// TIA Portal project "FactoryIO_Template_S7-1200_V16_V16" (V16)
// Vorlageprojekt für das Buch mit Zielsystem S7-1200

(* hardware
DEVICE "S7-1200-Station_1"  S7-1200 Station
   slot 0: "Baugruppenträger_0"  Rack  V1.0
   slot 1: "PLC_1"  CPU 1211C DC/DC/DC  6ES7 211-1AE40-0XB0  V4.1
*)

// ===== PLC "PLC_1"  CPU 1211C DC/DC/DC =====

VAR_GLOBAL   // PLC tag table "Standard-Variablentabelle"
   "Tag_1" AT %M0.0 : Bool;
   "Tag_2" AT %M0.1 : Bool;
   "Tag_3" AT %M0.2 : Bool;
   "Tag_4" AT %M0.3 : Bool;
   "Tag_5" AT %M0.4 : Bool;
   "Tag_6" AT %M0.5 : Bool;
   "Tag_7" AT %M1.0 : Bool;
   "Tag_8" AT %M0.6 : Bool;
   "Tag_9" AT %M1.2 : Bool;
   "Tag_10" AT %M1.5 : Bool;
   "Tag_11" AT %M0.7 : Bool;
END_VAR

VAR_GLOBAL   // PLC tag table "Tag table_1"
   "start" AT %I0.0 : Bool;
   "stop" AT %I0.1 : Bool;
   "sen 1" AT %I0.2 : Bool;
   "sen2" AT %I0.3 : Bool;
   "sen 3" AT %I0.4 : Bool;
   "sen4" AT %I0.5 : Bool;
   "sen 5" AT %I0.6 : Bool;
   "detect" AT %I0.7 : Bool;
   "X moving" AT %I1.0 : Bool;
   "Z moving" AT %I1.1 : Bool;
   "curve" AT %Q0.0 : Bool;
   "belt 4" AT %Q0.1 : Bool;
   "belt 6" AT %Q0.2 : Bool;
   "X" AT %Q0.3 : Bool;
   "Z" AT %Q0.4 : Bool;
   "grab" AT %Q0.5 : Bool;
END_VAR

FUNCTION "MHJ-PLC-Lab-Function-S71200" : Void   // FC9000, SCL
{ S7_Optimized_Access := 'TRUE' }
VERSION : 0.1
   VAR_TEMP
      rdTimeReturn : Int;
      outputTime : DTL;
      SyncVal : Byte;
      forVal : Int;
      forVal_2 : Int;
      Value : Byte;
   END_VAR
   VAR CONSTANT
      CompVal : Byte := 16#34;
      Value_01 : Byte := 16#11;
      Value_01_DW : DWord := 16#A165_D992;
      Value_02_DW : DWord := 16#58BE_4401;
   END_VAR
BEGIN

   #Value:=PEEK(area := 16#82,
        dbNumber := 0,
        byteOffset := 511);
   #Value := #Value + 1;

   POKE(area := 16#82,
        dbNumber := 0,
        byteOffset := 511,
        value := #Value);

   POKE(area:=16#81,
        dbNumber:=0,
        byteOffset:=1016,
        value:=#Value_01_DW);
   POKE(area := 16#81,
        dbNumber := 0,
        byteOffset := 1020,
        value := #Value_02_DW);

   POKE(area := 16#81,
        dbNumber := 0,
        byteOffset := 511,
        value := B#16#00);

   FOR #forVal := 0 TO 120 DO
       FOR #forVal_2:=0 TO 10 DO
           #rdTimeReturn:=RD_SYS_T(#outputTime);
           #rdTimeReturn := WR_SYS_T(#outputTime);
           #rdTimeReturn := RD_SYS_T(#outputTime);
           #rdTimeReturn := WR_SYS_T(#outputTime);
       END_FOR;
       #SyncVal:= PEEK(area := 16#81,
                      dbNumber := 0,
                      byteOffset := 511);
       IF #SyncVal = #CompVal THEN
          GOTO M_1;
       END_IF;
   END_FOR;
   RETURN;

   M_1:
   POKE(area := 16#81,
        dbNumber := 0,
        byteOffset := 511,
        value := B#16#0);
END_FUNCTION

ORGANIZATION_BLOCK "Main"   // OB1, LAD, ProgramCycle
TITLE = "Main Program Sweep (Cycle)"
{ S7_Optimized_Access := 'TRUE' }
VERSION : 0.1
   VAR_INPUT
      Initial_Call : Bool;   // Initial call of this OB
      Remanence : Bool;   // =True, if remanent data are available
   END_VAR
   VAR_TEMP   // added for the SCL form of the ladder/FBD networks
      _w1 : Bool;
   END_VAR
BEGIN

REGION Network 1: Konnektierungsbaustein für PLC-Lab
   // Im Netzwerk 1 wird der Konnektierungsbaustein für PLC-Lab aufgerufen.
   // Dieser Aufruf darf nicht entfernt werden!
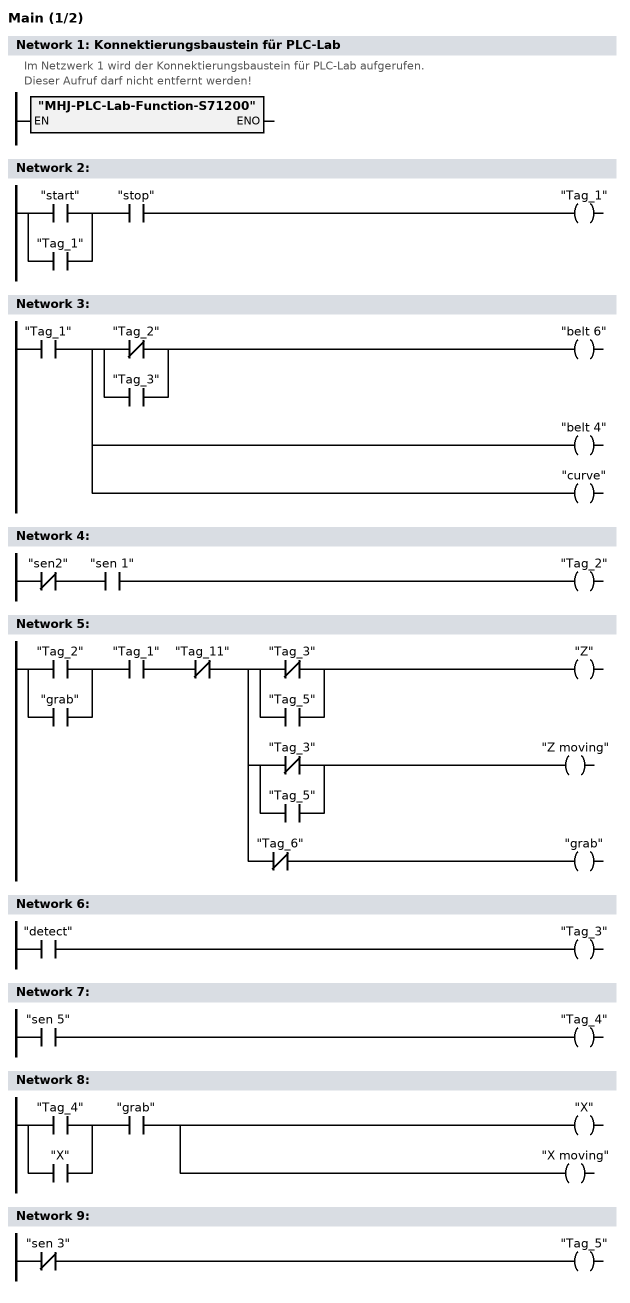
   RUNG wire#powerrail
      "MHJ-PLC-Lab-Function-S71200"()
   END_RUNG
   // the same network as SCL:
   "MHJ-PLC-Lab-Function-S71200"();
END_REGION

REGION Network 2
   RUNG wire#powerrail
      Contact( "start" )
      wire#w1
      Contact( "stop" )
      Coil( "Tag_1" )
   END_RUNG
   RUNG wire#powerrail
      Contact( "Tag_1" )
   END_RUNG wire#w1
   // the same network as SCL:
   "Tag_1" := ("start" OR "Tag_1") AND "stop";
END_REGION

REGION Network 3
   RUNG wire#powerrail
      Contact( "Tag_1" )
      wire#w1
      I_Contact( "Tag_2" )
      wire#w2
      Coil( "belt 6" )
   END_RUNG
   RUNG wire#w1
      Contact( "Tag_3" )
   END_RUNG wire#w2
   RUNG wire#w1
      Coil( "belt 4" )
   END_RUNG
   RUNG wire#w1
      Coil( "curve" )
   END_RUNG
   // the same network as SCL:
   "belt 6" := "Tag_1" AND (NOT "Tag_2" OR "Tag_3");
   "belt 4" := "Tag_1";
   "curve" := "Tag_1";
END_REGION

REGION Network 4
   RUNG wire#powerrail
      I_Contact( "sen2" )
      Contact( "sen 1" )
      Coil( "Tag_2" )
   END_RUNG
   // the same network as SCL:
   "Tag_2" := NOT "sen2" AND "sen 1";
END_REGION

REGION Network 5
   RUNG wire#powerrail
      Contact( "Tag_2" )
      wire#w1
      Contact( "Tag_1" )
      I_Contact( "Tag_11" )
      wire#w2
      I_Contact( "Tag_3" )
      wire#w3
      Coil( "Z" )
   END_RUNG
   RUNG wire#powerrail
      Contact( "grab" )
   END_RUNG wire#w1
   RUNG wire#w2
      Contact( "Tag_5" )
   END_RUNG wire#w3
   RUNG wire#w2
      I_Contact( "Tag_3" )
      wire#w4
      Coil( "Z moving" )
   END_RUNG
   RUNG wire#w2
      Contact( "Tag_5" )
   END_RUNG wire#w4
   RUNG wire#w2
      I_Contact( "Tag_6" )
      Coil( "grab" )
   END_RUNG
   // the same network as SCL:
   #_w1 := ("Tag_2" OR "grab") AND "Tag_1" AND NOT "Tag_11";
   "Z" := #_w1 AND (NOT "Tag_3" OR "Tag_5");
   "Z moving" := #_w1 AND (NOT "Tag_3" OR "Tag_5");
   "grab" := #_w1 AND NOT "Tag_6";
END_REGION

REGION Network 6
   RUNG wire#powerrail
      Contact( "detect" )
      Coil( "Tag_3" )
   END_RUNG
   // the same network as SCL:
   "Tag_3" := "detect";
END_REGION

REGION Network 7
   RUNG wire#powerrail
      Contact( "sen 5" )
      Coil( "Tag_4" )
   END_RUNG
   // the same network as SCL:
   "Tag_4" := "sen 5";
END_REGION

REGION Network 8
   RUNG wire#powerrail
      Contact( "Tag_4" )
      wire#w1
      Contact( "grab" )
      wire#w2
      Coil( "X" )
   END_RUNG
   RUNG wire#powerrail
      Contact( "X" )
   END_RUNG wire#w1
   RUNG wire#w2
      Coil( "X moving" )
   END_RUNG
   // the same network as SCL:
   "X" := ("Tag_4" OR "X") AND "grab";
   "X moving" := "X";
END_REGION

REGION Network 9
   RUNG wire#powerrail
      I_Contact( "sen 3" )
      Coil( "Tag_5" )
   END_RUNG
   // the same network as SCL:
   "Tag_5" := NOT "sen 3";
END_REGION

REGION Network 10
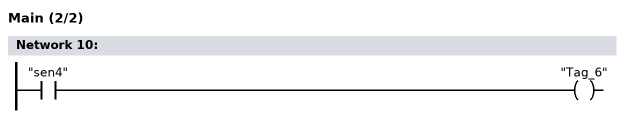
   RUNG wire#powerrail
      Contact( "sen4" )
      Coil( "Tag_6" )
   END_RUNG
   // the same network as SCL:
   "Tag_6" := "sen4";
END_REGION
END_ORGANIZATION_BLOCK